// Mitsubishi GX Works2 project: 4   PLC: FX2N/FX2NC

PROGRAM MAIN
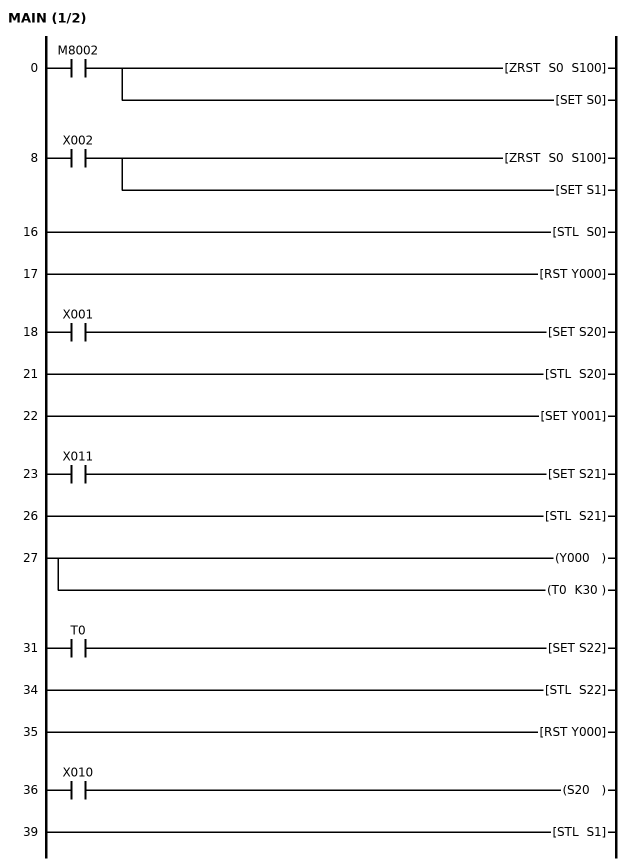
0     LD      M8002
      ZRST    S0 S100
      SET     S0
8     LD      X002
      ZRST    S0 S100
      SET     S1
16    STL     S0
17    RST     Y000
18    LD      X001
      SET     S20
21    STL     S20
22    SET     Y001
23    LD      X011
      SET     S21
26    STL     S21
27    OUT     Y000
      OUT     T0 K30
31    LD      T0
      SET     S22
34    STL     S22
35    RST     Y000
36    LD      X010
      OUT     S20
39    STL     S1
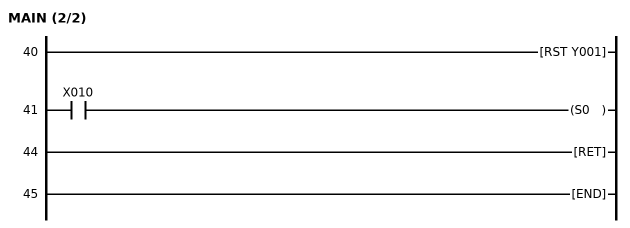
40    RST     Y001
41    LD      X010
      OUT     S0
44    RET
45    END
END_PROGRAM

// device comments not shown above
BL0  ; main
BL1  ; a
BL2  ; b
